FUNCTION_BLOCK FB_MotorControl
VAR_INPUT
	Button1 : BOOL;
	Button2 : BOOL;
	Sensor : BOOL;
END_VAR
VAR_OUTPUT
	Motor : BOOL;
END_VAR
VAR
END_VAR

Motor := IsMotorTurnedOn(Button1, Button2, Sensor);

METHOD IsMotorTurnedOn : BOOL
VAR_INPUT
	button1 : BOOL;
	button2 : BOOL;
	sensor : bool;
END_VAR
IsMotorTurnedOn := button1 AND button2 AND NOT sensor;
END_METHOD

END_FUNCTION_BLOCK

(* stored: Version 1.1.0.1, ProductVersion 3.1.4024.12
   POU FB_MotorControl: Id {baa4aa47-6872-434b-b7d0-1f178110ceec}, SpecialFunc None
   Method IsMotorTurnedOn: Id {458f2903-6a68-4aab-b843-bb1060e63ef3} *)
